TYPE T_NEST_OFFSET : ARRAY[1..MAX_MOVER]        OF
                     ARRAY[1..MAX_STATION_NEST] OF LREAL;
END_TYPE

(* stored: Version 1.1.0.1, ProductVersion 3.1.4026.18
   DUT T_NEST_OFFSET: Id {b40e6ee2-e3ad-4c06-937e-5cf91a5cbc5d} *)
